(* IEC 61131-3 sources: CS-6263/cs_6263_mp_2/amd/Solutions_p1/part1c/build, 2 files *)

(* ---- plc.st ---- *)
TYPE
  LOGLEVEL : (CRITICAL, WARNING, INFO, DEBUG) := INFO;
END_TYPE

FUNCTION_BLOCK LOGGER
  VAR_INPUT
    TRIG : BOOL;
    MSG : STRING;
    LEVEL : LOGLEVEL := INFO;
  END_VAR
  VAR
    TRIG0 : BOOL;
  END_VAR

  IF TRIG AND NOT TRIG0 THEN
  {{
   LogMessage(GetFbVar(LEVEL),(char*)GetFbVar(MSG, .body),GetFbVar(MSG, .len));
  }}
  END_IF;
  TRIG0:=TRIG;
END_FUNCTION_BLOCK

PROGRAM part1c
  VAR
    Input0 : BOOL;
    Output0 : BOOL;
  END_VAR
  VAR
    Oscillator : BOOL;
    TON0 : TON;
    TOF0 : TOF;
    CTU0 : CTU;
    Bomb : BOOL;
    Countup : INT := 6;
    TrueBool : BOOL := 1;
    TON1 : TON;
    R_TRIG1 : R_TRIG;
  END_VAR

  TON0(IN := NOT(Oscillator) AND Input0, PT := T#6000ms);
  TOF0(IN := TON0.Q, PT := T#6000ms);
  Oscillator := TOF0.Q;
  Output0 := Bomb OR NOT(Oscillator) AND Input0;
  R_TRIG1(CLK := Output0);
  CTU0(CU := R_TRIG1.Q, PV := Countup);
  TON1(IN := Input0, PT := T#30000ms);
  Bomb := Bomb OR CTU0.Q OR TON1.Q;
END_PROGRAM

CONFIGURATION Config0

  RESOURCE Res0 ON PLC
    TASK task0(INTERVAL := T#20ms,PRIORITY := 0);
    PROGRAM instance0 WITH task0 : part1c;
  END_RESOURCE
END_CONFIGURATION

(* ---- generated_plc.st ---- *)
PROGRAM part1c
  VAR
    Input0 AT %IX1.0 : BOOL;
    Output0 AT %QX1.0 : BOOL;
  END_VAR
  VAR
    Oscillator : BOOL;
    TON0 : TON;
    TOF0 : TOF;
    CTU0 : CTU;
    Bomb : BOOL;
    Countup : INT := 6;
    TrueBool : BOOL := 1;
    TON1 : TON;
    R_TRIG1 : R_TRIG;
  END_VAR

  TON0(IN := NOT(Oscillator) AND Input0, PT := T#6000ms);
  TOF0(IN := TON0.Q, PT := T#6000ms);
  Oscillator := TOF0.Q;
  Output0 := Bomb OR NOT(Oscillator) AND Input0;
  R_TRIG1(CLK := Output0);
  CTU0(CU := R_TRIG1.Q, PV := Countup);
  TON1(IN := Input0, PT := T#30000ms);
  Bomb := Bomb OR CTU0.Q OR TON1.Q;
END_PROGRAM

CONFIGURATION Config0

  RESOURCE Res0 ON PLC
    TASK task0(INTERVAL := T#20ms,PRIORITY := 0);
    PROGRAM instance0 WITH task0 : part1c;
  END_RESOURCE
END_CONFIGURATION
